# B&R Automation Studio project A2019059_Linka_Power_CP (part 39)

#### Main.st - Init, cyclic, exit code
```iecst
PROGRAM _INIT
	P34_Vizu.GoPage:= 'PageBootP34';

END_PROGRAM

PROGRAM _CYCLIC

	//************************************Filter alarmov**************************************************************//
	FilterVizu_P34:= '[{"logicalOperator":"and","value":300,"conditionType":">=","columnType":"cod","useAlarmState":false,"alarmState":0},{"value":500,"conditionType":"<=","columnType":"cod","useAlarmState":false,"alarmState":0}]';

	//***********************************Zobrazenie warningov pracoviska 3****************************************************//
	//0 - Pracovisko je vypnuté.
	//1 - Prebieha inicializácia pracoviska.
	//2 - Na pracovisku prebieha výroba.
	//3 - Prebieha ukončenie pracovného cyklu pracoviska.
	//4 - Prebieha režim vyprázdnenia linky.
	//5 - Doplň zásobník skrutiek K40 !!!
	//6 - Doplň zásobník skrutiek M5 !!!
	//7 - Niesu založené správne kontakty na HV teste !!!
	//8 - Niesu založené správne kontakty na Leakage teste stanica A !!!
	//9 - Niesu založené správne kontakty na Leakage teste stanica B !!!

	IF Linka.PAR.ZvolenyModel = '4F' AND NOT P3_Srobovanie.IN.HVTest_TypKonektoru_4F THEN
		P34_Vizu.WarningsP3_Index:= 7;
	ELSIF Linka.PAR.ZvolenyModel = '5F' AND NOT P3_Srobovanie.IN.HVTest_TypKonektoru_5F_5H THEN
		P34_Vizu.WarningsP3_Index:= 7;
	ELSIF Linka.PAR.ZvolenyModel = '5H' AND NOT P3_Srobovanie.IN.HVTest_TypKonektoru_5F_5H THEN
		P34_Vizu.WarningsP3_Index:= 7;
	ELSIF Linka.PAR.ZvolenyModel = '4F' AND NOT P3_LeakageTestA.IN.Tester_TypKonektoru_4F THEN
		P34_Vizu.WarningsP3_Index:= 8;
	ELSIF Linka.PAR.ZvolenyModel = '5F' AND NOT P3_LeakageTestA.IN.Tester_TypKonektoru_5F_5H THEN
		P34_Vizu.WarningsP3_Index:= 8;
	ELSIF Linka.PAR.ZvolenyModel = '5H' AND NOT P3_LeakageTestA.IN.Tester_TypKonektoru_5F_5H THEN
		P34_Vizu.WarningsP3_Index:= 8;
	ELSIF Linka.PAR.ZvolenyModel = '4F' AND NOT P3_LeakageTestB.IN.Tester_TypKonektoru_4F THEN
		P34_Vizu.WarningsP3_Index:= 9;
	ELSIF Linka.PAR.ZvolenyModel = '5F' AND NOT P3_LeakageTestB.IN.Tester_TypKonektoru_5F_5H THEN
		P34_Vizu.WarningsP3_Index:= 9;
	ELSIF Linka.PAR.ZvolenyModel = '5H' AND NOT P3_LeakageTestB.IN.Tester_TypKonektoru_5F_5H THEN
		P34_Vizu.WarningsP3_Index:= 9;
	ELSIF P3_Srobovanie.STAV.Zasobnik_K40_Prazdny THEN
		P34_Vizu.WarningsP3_Index:= 5;
	ELSIF P3_Srobovanie.STAV.Zasobnik_M5_Prazdny THEN
        P34_Vizu.WarningsP3_Index:= 6;
    ELSIF Linka.TestovaciKus THEN
        P34_Vizu.WarningsP3_Index:= 11;
	ELSIF Linka.VyprazdnenieLinky THEN
		P34_Vizu.WarningsP3_Index:= 4;
	ELSIF P3_Pracovisko.STAV.Automat AND NOT P3_Pracovisko.STAV.PoINIT AND NOT P3_Pracovisko.STAV.UkoncenieCyklu_BUSY THEN
		P34_Vizu.WarningsP3_Index:= 1;
	ELSIF P3_Pracovisko.STAV.PoINIT AND NOT P3_Pracovisko.STAV.UkoncenieCyklu_BUSY THEN
		P34_Vizu.WarningsP3_Index:= 2;
	ELSIF P3_Pracovisko.STAV.UkoncenieCyklu_BUSY THEN
		P34_Vizu.WarningsP3_Index:= 3;
	ELSIF NOT P3_Pracovisko.STAV.Automat THEN
		P34_Vizu.WarningsP3_Index:= 0;
	END_IF

	P34_Vizu.WarningsP3_Index;

	//************************Prepínanie farby textového pola warning pracoviska 3***********************************//
	IF P34_Vizu.WarningsP3_Index = 0 THEN
		P34_Vizu.WarningsP3_Farba:= "TextOutput_Green";
	ELSIF P34_Vizu.WarningsP3_Index = 1 THEN
		P34_Vizu.WarningsP3_Farba:= "TextOutput_Green";
	ELSIF P34_Vizu.WarningsP3_Index = 2 THEN
		P34_Vizu.WarningsP3_Farba:= "TextOutput_Green";
	ELSIF P34_Vizu.WarningsP3_Index = 3 THEN
		P34_Vizu.WarningsP3_Farba:= "TextOutput_Green";
	ELSIF P34_Vizu.WarningsP3_Index = 4 THEN
        P34_Vizu.WarningsP3_Farba:= "TextOutput_Green";
    ELSIF P34_Vizu.WarningsP3_Index = 11 THEN
        P34_Vizu.WarningsP3_Farba:= "TextOutput_Green";
	ELSE
		IF Blikac1s THEN
			P34_Vizu.WarningsP3_Farba:= "TextOutput_Red";
		ELSE
			P34_Vizu.WarningsP3_Farba:= "TextOutput_Grey";
		END_IF
	END_IF

	//***********************************Zobrazenie warningov pracoviska 4****************************************************//
	//0 - Pracovisko je vypnuté.
	//1 - Prebieha inicializácia pracoviska.
	//2 - Na pracovisku prebieha výroba.
	//3 - Prebieha ukončenie pracovného cyklu pracoviska.
	//4 - Prebieha režim vyprázdnenia linky.
	//5 - Niesu založené správne kontakty na Funkčnom teste stanica A !!!
	//6 - Niesu založené správne kontakty na Funkčnom teste stanica B !!!

	IF Linka.PAR.ZvolenyModel = '4F' AND NOT P4_FunkcnyTestA.IN.TypSpodnychKontaktov_4F THEN
		P34_Vizu.WarningsP4_Index:= 5;
	ELSIF Linka.PAR.ZvolenyModel = '5F' AND NOT P4_FunkcnyTestA.IN.TypSpodnychKontaktov_5F_5H THEN
		P34_Vizu.WarningsP4_Index:= 5;
	ELSIF Linka.PAR.ZvolenyModel = '5H' AND NOT P4_FunkcnyTestA.IN.TypSpodnychKontaktov_5F_5H THEN
		P34_Vizu.WarningsP4_Index:= 5;
	ELSIF Linka.PAR.ZvolenyModel = '4F' AND NOT P4_FunkcnyTestB.IN.TypSpodnychKontaktov_4F THEN
		P34_Vizu.WarningsP4_Index:= 6;
	ELSIF Linka.PAR.ZvolenyModel = '5F' AND NOT P4_FunkcnyTestB.IN.TypSpodnychKontaktov_5F_5H THEN
		P34_Vizu.WarningsP4_Index:= 6;
	ELSIF Linka.PAR.ZvolenyModel = '5H' AND NOT P4_FunkcnyTestB.IN.TypSpodnychKontaktov_5F_5H THEN
        P34_Vizu.WarningsP4_Index:= 6;
    ELSIF Linka.TestovaciKus THEN
        P34_Vizu.WarningsP4_Index:= 8;
	ELSIF Linka.VyprazdnenieLinky THEN
		P34_Vizu.WarningsP4_Index:= 4;
	ELSIF P4_Pracovisko.STAV.Automat AND NOT P4_Pracovisko.STAV.PoINIT AND NOT P4_Pracovisko.STAV.UkoncenieCyklu_BUSY THEN
		P34_Vizu.WarningsP4_Index:= 1;
	ELSIF P4_Pracovisko.STAV.PoINIT AND NOT P4_Pracovisko.STAV.UkoncenieCyklu_BUSY THEN
		P34_Vizu.WarningsP4_Index:= 2;
	ELSIF P4_Pracovisko.STAV.UkoncenieCyklu_BUSY THEN
		P34_Vizu.WarningsP4_Index:= 3;
	ELSIF NOT P4_Pracovisko.STAV.Automat THEN
		P34_Vizu.WarningsP4_Index:= 0;
	END_IF

	//************************Prepínanie farby textového pola warning pracoviska 4***********************************//
	IF P34_Vizu.WarningsP4_Index = 0 THEN
		P34_Vizu.WarningsP4_Farba:= "TextOutput_Green";
	ELSIF P34_Vizu.WarningsP4_Index = 1 THEN
		P34_Vizu.WarningsP4_Farba:= "TextOutput_Green";
	ELSIF P34_Vizu.WarningsP4_Index = 2 THEN
		P34_Vizu.WarningsP4_Farba:= "TextOutput_Green";
	ELSIF P34_Vizu.WarningsP4_Index = 3 THEN
		P34_Vizu.WarningsP4_Farba:= "TextOutput_Green";
	ELSIF P34_Vizu.WarningsP4_Index = 4 THEN
        P34_Vizu.WarningsP4_Farba:= "TextOutput_Green";
    ELSIF P34_Vizu.WarningsP4_Index = 8 THEN
        P34_Vizu.WarningsP4_Farba:= "TextOutput_Green";
	ELSE
		IF Blikac1s THEN
			P34_Vizu.WarningsP4_Farba:= "TextOutput_Red";
		ELSE
			P34_Vizu.WarningsP4_Farba:= "TextOutput_Grey";
		END_IF
	END_IF

	//***********************Prepnutie na obrazovku Automat z ručného režimu******************//
    IF P3_Pracovisko.STAV.Manual AND NOT Safety.STAV.P3_ZamkyBunky_AKTIVNE THEN
        P3_Pracovisko.Reset:= TRUE;
        P34_Vizu.GoPage:= 'PageBootP34';
    END_IF
    IF P4_Pracovisko.STAV.Manual AND NOT Safety.STAV.P4_ZamkyBunky_AKTIVNE THEN
        P4_Pracovisko.Reset:= TRUE;
        P34_Vizu.GoPage:= 'PageBootP34';
    END_IF

	//***********************Prepnutie bootovacej obrazovky********************************//
	IF NOT Safety.STAV.SafetyPLC_Nabehlo THEN
        P34_Vizu.GoPage:= 'PageBootP34';
    ELSIF CasPrepnutiaObrazovky.Q THEN
        P34_Vizu.GoPage:= 'PageBootP34';
	ELSIF P34_Vizu.ActualPage = 'PageBootP34' AND Safety.STAV.SafetyPLC_Nabehlo THEN
		P34_Vizu.GoPage:= 'PageAutomatP34';
	END_IF

    CasPrepnutiaObrazovky.IN:= P34_Vizu.ActualPage = 'PageBootP34' AND P34_Vizu.GoPage = 'PageAutomatP34';
    CasPrepnutiaObrazovky.PT:= T#5s;
    CasPrepnutiaObrazovky();

    //**************************Zamknutie editácie parametrov *********************************//

    IF P34_UrovenPrihlasenehoUzivatela >= 20 THEN
        P34_Vizu.EditaciaParametrov_ENABLE:= TRUE;
    ELSE
        P34_Vizu.EditaciaParametrov_ENABLE:= FALSE;
    END_IF

	//*************************************Zamknutie tlačítok - Pracovisko 3***************************************************************//
	//Tlačítko Štat Automat //
	IF P3_Pracovisko.STAV.UkoncenieCyklu_BUSY THEN
		P34_Vizu.TL_StartAutomat_ENABLE_P3:= FALSE;
	ELSIF P3_Pracovisko.STAV.PORUCHA THEN
		P34_Vizu.TL_StartAutomat_ENABLE_P3:= FALSE;
	ELSIF Linka.PAR.ZvolenyModel = '4F' AND NOT P3_Srobovanie.IN.HVTest_TypKonektoru_4F THEN
		P34_Vizu.TL_StartAutomat_ENABLE_P3:= FALSE;
	ELSIF Linka.PAR.ZvolenyModel = '5F' AND NOT P3_Srobovanie.IN.HVTest_TypKonektoru_5F_5H THEN
		P34_Vizu.TL_StartAutomat_ENABLE_P3:= FALSE;
	ELSIF Linka.PAR.ZvolenyModel = '5H' AND NOT P3_Srobovanie.IN.HVTest_TypKonektoru_5F_5H THEN
		P34_Vizu.TL_StartAutomat_ENABLE_P3:= FALSE;
	ELSIF Linka.PAR.ZvolenyModel = '4F' AND NOT P3_LeakageTestA.IN.Tester_TypKonektoru_4F THEN
		P34_Vizu.TL_StartAutomat_ENABLE_P3:= FALSE;
	ELSIF Linka.PAR.ZvolenyModel = '5F' AND NOT P3_LeakageTestA.IN.Tester_TypKonektoru_5F_5H THEN
		P34_Vizu.TL_StartAutomat_ENABLE_P3:= FALSE;
	ELSIF Linka.PAR.ZvolenyModel = '5H' AND NOT P3_LeakageTestA.IN.Tester_TypKonektoru_5F_5H THEN
		P34_Vizu.TL_StartAutomat_ENABLE_P3:= FALSE;
	ELSIF Linka.PAR.ZvolenyModel = '4F' AND NOT P3_LeakageTestB.IN.Tester_TypKonektoru_4F THEN
		P34_Vizu.TL_StartAutomat_ENABLE_P3:= FALSE;
	ELSIF Linka.PAR.ZvolenyModel = '5F' AND NOT P3_LeakageTestB.IN.Tester_TypKonektoru_5F_5H THEN
		P34_Vizu.TL_StartAutomat_ENABLE_P3:= FALSE;
	ELSIF Linka.PAR.ZvolenyModel = '5H' AND NOT P3_LeakageTestB.IN.Tester_TypKonektoru_5F_5H THEN
		P34_Vizu.TL_StartAutomat_ENABLE_P3:= FALSE;
	ELSIF NOT Safety.STAV.P3_ZonaBunky_AKTIVNA THEN
		P34_Vizu.TL_StartAutomat_ENABLE_P3:= FALSE;
	ELSE
		P34_Vizu.TL_StartAutomat_ENABLE_P3:= TRUE;
	END_IF

	//Tlačítko Ukončenie Cyklu//
	IF P3_Pracovisko.STAV.PoINIT THEN
		P34_Vizu.TL_KoniecCyklu_ENABLE_P3:= TRUE;
	ELSE
		P34_Vizu.TL_KoniecCyklu_ENABLE_P3:= FALSE;
	END_IF

    //Tlačítko STOP//
    IF P3_Pracovisko.STAV.PoINIT THEN
        P34_Vizu.TL_STOP_ENABLE_P3:= FALSE;
    ELSE
        P34_Vizu.TL_STOP_ENABLE_P3:= TRUE;
    END_IF

	//Tlačítko Režim Automat//

	P34_Vizu.TL_RezimAutomat_ENABLE:= TRUE;

	//Tlačítko Režim Manual - pracovisko 3//
	IF P3_Pracovisko.STAV.Automat THEN
		P34_Vizu.TL_RezimManual_ENABLE_P3:= FALSE;
	ELSIF NOT P3_Pracovisko.STAV.Manual AND NOT P3_Pracovisko.STAV.READY THEN
		P34_Vizu.TL_RezimManual_ENABLE_P3:= FALSE;
	ELSIF NOT Safety.STAV.P3_ZamkyBunky_AKTIVNE THEN
        P34_Vizu.TL_RezimManual_ENABLE_P3:= FALSE;
    ELSE
		P34_Vizu.TL_RezimManual_ENABLE_P3:= TRUE;
	END_IF

    //Tlačítka ovládania zámkov//
    IF NOT P3_Pracovisko.STAV.Automat THEN
        P34_Vizu.TL_OvladaniaZamkov_ENABLE_P3:= TRUE;
    ELSE
        P34_Vizu.TL_OvladaniaZamkov_ENABLE_P3:= FALSE;
    END_IF

    //Volba zapnutia Leakage Testu//
    IF P3_Pracovisko.STAV.Automat THEN
        P34_Vizu.VolbaLeakageTestu_ENABLE:= FALSE;
    ELSE
        P34_Vizu.VolbaLeakageTestu_ENABLE:= TRUE;
    END_IF

    //Tlačítka spustenie čistenie skrutkovačiek v ručnom režime//
    IF NOT P3_Srobovacky_VychodziaPozicia THEN
        P34_Vizu.RR_CistenieSkrutkovaciek_ENABLE:= FALSE;
    ELSIF P3_Srobovanie.STAV.Cistenie_K40_BUSY THEN
        P34_Vizu.RR_CistenieSkrutkovaciek_ENABLE:= FALSE;
    ELSIF NOT P3_Srobovanie.STAV.OsY_HomingOK THEN
        P34_Vizu.RR_CistenieSkrutkovaciek_ENABLE:= FALSE;
    ELSIF P34_UrovenPrihlasenehoUzivatela < 20 THEN
        P34_Vizu.RR_CistenieSkrutkovaciek_ENABLE:= FALSE;
    ELSIF P3_Srobovanie.RR_PolohujNaPoziciuSkrutky_4F5F THEN
        P34_Vizu.RR_CistenieSkrutkovaciek_ENABLE:= FALSE;
    ELSIF P3_Srobovanie.RR_PolohujNaPoziciuSkrutky_5H THEN
        P34_Vizu.RR_CistenieSkrutkovaciek_ENABLE:= FALSE;
    ELSE
        P34_Vizu.RR_CistenieSkrutkovaciek_ENABLE:= TRUE;
    END_IF

    //Tlačítka ovládania osy Y manipulatora šróbovačiek//
    IF NOT P3_Srobovanie.STAV.OsY_HomingOK THEN
        P34_Vizu.Srobovanie_OvlManipOsY_ENABLE:= FALSE;
    ELSIF NOT P3_Srobovacky_VychodziaPozicia THEN
        P34_Vizu.Srobovanie_OvlManipOsY_ENABLE:= FALSE;
    ELSIF P3_Srobovanie.RR_PolohujNaPoziciuSkrutky_4F5F THEN
        P34_Vizu.Srobovanie_OvlManipOsY_ENABLE:= FALSE;
    ELSIF P3_Srobovanie.RR_PolohujNaPoziciuSkrutky_5H THEN
        P34_Vizu.Srobovanie_OvlManipOsY_ENABLE:= FALSE;
    ELSIF P3_Srobovanie.STAV.Cistenie_K40_BUSY THEN
        P34_Vizu.Srobovanie_OvlManipOsY_ENABLE:= FALSE;
    ELSE
        P34_Vizu.Srobovanie_OvlManipOsY_ENABLE:= TRUE;
    END_IF

    //Zamknutie tlačítok test pozicii skrutkovačiek//
    IF NOT P3_Srobovanie.STAV.OsY_HomingOK THEN
        P34_Vizu.RR_PozicieSkrutiek_ENABLE:= FALSE;
    ELSIF NOT P3_Srobovacky_VychodziaPozicia THEN
        P34_Vizu.RR_PozicieSkrutiek_ENABLE:= FALSE;
    ELSIF P3_Srobovanie.STAV.Cistenie_K40_BUSY THEN
        P34_Vizu.RR_PozicieSkrutiek_ENABLE:= FALSE;
    ELSIF P34_UrovenPrihlasenehoUzivatela < 100 THEN
        P34_Vizu.RR_PozicieSkrutiek_ENABLE:= FALSE;
    ELSIF P3_Srobovanie.RR_PolohujNaPoziciuSkrutky_4F5F THEN
        P34_Vizu.RR_PozicieSkrutiek_ENABLE:= FALSE;
    ELSIF P3_Srobovanie.RR_PolohujNaPoziciuSkrutky_5H THEN
        P34_Vizu.RR_PozicieSkrutiek_ENABLE:= FALSE;
    ELSE
        P34_Vizu.RR_PozicieSkrutiek_ENABLE:= TRUE;
    END_IF

    //Tlačítko testovania Leakage Testu A v ručnom režime//
    IF NOT Safety.STAV.P3_ZonaBunky_AKTIVNA THEN
        P34_Vizu.LeakageTestA_Testovanie_ENABLE:= FALSE;
    ELSIF NOT P3_LeakageTestA.IN.PritomnostPaletky_S23 THEN
       P34_Vizu.LeakageTestA_Testovanie_ENABLE:= FALSE;
    ELSE
        P34_Vizu.LeakageTestA_Testovanie_ENABLE:= TRUE;
    END_IF

    //Tlačítko testovania Leakage Testu B v ručnom režime//
    IF NOT Safety.STAV.P3_ZonaBunky_AKTIVNA THEN
        P34_Vizu.LeakageTestB_Testovanie_ENABLE:= FALSE;
    ELSIF NOT P3_LeakageTestB.IN.PritomnostPaletky_S24 THEN
        P34_Vizu.LeakageTestB_Testovanie_ENABLE:= FALSE;
    ELSE
        P34_Vizu.LeakageTestB_Testovanie_ENABLE:= TRUE;
    END_IF

    //Zamknutie tlačítok ovládania Leakage testu A v ručnom režime//
    IF P3_LeakageTestA.STAV.TestovaciaSekvencia_BUSY THEN
        P34_Vizu.LeakageTestA_RR_ENABLE:= FALSE;
    ELSE
        P34_Vizu.LeakageTestA_RR_ENABLE:= TRUE;
    END_IF

   //Zamknutie tlačítok ovládania Leakage testu B v ručnom režime//
    IF P3_LeakageTestB.STAV.TestovaciaSekvencia_BUSY THEN
        P34_Vizu.LeakageTestB_RR_ENABLE:= FALSE;
    ELSE
        P34_Vizu.LeakageTestB_RR_ENABLE:= TRUE;
    END_IF

	//*************************************Zamknutie tlačítok - Pracovisko 4***************************************************************//
	//Tlačítko Štat Automat//
	IF P4_Pracovisko.STAV.UkoncenieCyklu_BUSY THEN
		P34_Vizu.TL_StartAutomat_ENABLE_P4:= FALSE;
	ELSIF P4_Pracovisko.STAV.PORUCHA THEN
		P34_Vizu.TL_StartAutomat_ENABLE_P4:= FALSE;
	ELSIF Linka.PAR.ZvolenyModel = '4F' AND NOT P4_FunkcnyTestA.IN.TypSpodnychKontaktov_4F THEN
		P34_Vizu.TL_StartAutomat_ENABLE_P4:= FALSE;
	ELSIF Linka.PAR.ZvolenyModel = '5F' AND NOT P4_FunkcnyTestA.IN.TypSpodnychKontaktov_5F_5H THEN
		P34_Vizu.TL_StartAutomat_ENABLE_P4:= FALSE;
	ELSIF Linka.PAR.ZvolenyModel = '5H' AND NOT P4_FunkcnyTestA.IN.TypSpodnychKontaktov_5F_5H THEN
		P34_Vizu.TL_StartAutomat_ENABLE_P4:= FALSE;
	ELSIF Linka.PAR.ZvolenyModel = '4F' AND NOT P4_FunkcnyTestB.IN.TypSpodnychKontaktov_4F THEN
		P34_Vizu.TL_StartAutomat_ENABLE_P4:= FALSE;
	ELSIF Linka.PAR.ZvolenyModel = '5F' AND NOT P4_FunkcnyTestB.IN.TypSpodnychKontaktov_5F_5H THEN
		P34_Vizu.TL_StartAutomat_ENABLE_P4:= FALSE;
	ELSIF Linka.PAR.ZvolenyModel = '5H' AND NOT P4_FunkcnyTestB.IN.TypSpodnychKontaktov_5F_5H THEN
		P34_Vizu.TL_StartAutomat_ENABLE_P4:= FALSE;
	ELSIF NOT Safety.STAV.P4_ZonaBunky_AKTIVNA THEN
		P34_Vizu.TL_StartAutomat_ENABLE_P4:= FALSE;
	ELSE
		P34_Vizu.TL_StartAutomat_ENABLE_P4:= TRUE;
	END_IF

	//Tlačítko Ukončenie Cyklu//
	IF P4_Pracovisko.STAV.PoINIT THEN
		P34_Vizu.TL_KoniecCyklu_ENABLE_P4:= TRUE;
	ELSE
		P34_Vizu.TL_KoniecCyklu_ENABLE_P4:= FALSE;
	END_IF

    //Tlačítko STOP//
    IF P4_Pracovisko.STAV.PoINIT THEN
        P34_Vizu.TL_STOP_ENABLE_P4:= FALSE;
    ELSE
        P34_Vizu.TL_STOP_ENABLE_P4:= TRUE;
    END_IF

    //Tlačítko vyprázdnenie linky//
    IF Linka.VyprazdnenieLinky THEN
        P34_Vizu.TL_VyprazdnenieLinky_ENABLE:= FALSE;
    ELSIF NOT P4_Pracovisko.STAV.Automat THEN
        P34_Vizu.TL_VyprazdnenieLinky_ENABLE:= FALSE;
    ELSIF Linka.TestovaciKus THEN
        P34_Vizu.TL_VyprazdnenieLinky_ENABLE:= FALSE;
    ELSE
        P34_Vizu.TL_VyprazdnenieLinky_ENABLE:= TRUE;
    END_IF

	//Tlačítka ovládania zámkov//
	IF NOT P4_Pracovisko.STAV.Automat THEN
		P34_Vizu.TL_OvladaniaZamkov_ENABLE_P4:= TRUE;
	ELSE
		P34_Vizu.TL_OvladaniaZamkov_ENABLE_P4:= FALSE;
	END_IF

    //Tlačítko Režim Manual - pracovisko 4//
    IF P4_Pracovisko.STAV.Automat THEN
        P34_Vizu.TL_RezimManual_ENABLE_P4:= FALSE;
    ELSIF NOT P4_Pracovisko.STAV.Manual AND NOT P4_Pracovisko.STAV.READY THEN
        P34_Vizu.TL_RezimManual_ENABLE_P4:= FALSE;
    ELSIF NOT Safety.STAV.P4_ZamkyBunky_AKTIVNE THEN
        P34_Vizu.TL_RezimManual_ENABLE_P4:= FALSE;
    ELSE
        P34_Vizu.TL_RezimManual_ENABLE_P4:= TRUE;
    END_IF

    //Volba zapnutia Funkčného Testu//
    IF P4_Pracovisko.STAV.Automat THEN
        P34_Vizu.VolbaFunkcnehoTestu_ENABLE:= FALSE;
    ELSE
        P34_Vizu.VolbaFunkcnehoTestu_ENABLE:= TRUE;
    END_IF

    //Tlačítko testovania Funkčného Testu A v ručnom režime//
    IF NOT Safety.STAV.P4_ZonaBunky_AKTIVNA THEN
        P34_Vizu.FunkcnyTestA_Testovanie_ENABLE:= FALSE;
    ELSIF NOT P4_FunkcnyTestA.IN.PritomnostPaletky_S10 THEN
        P34_Vizu.FunkcnyTestA_Testovanie_ENABLE:= FALSE;
    ELSE
        P34_Vizu.FunkcnyTestA_Testovanie_ENABLE:= TRUE;
    END_IF

    //Tlačítko testovania Funkčného Testu B v ručnom režime//
    IF NOT Safety.STAV.P4_ZonaBunky_AKTIVNA THEN
        P34_Vizu.FunkcnyTestB_Testovanie_ENABLE:= FALSE;
    ELSIF NOT P4_FunkcnyTestB.IN.PritomnostPaletky_S11 THEN
        P34_Vizu.FunkcnyTestB_Testovanie_ENABLE:= FALSE;
    ELSE
        P34_Vizu.FunkcnyTestB_Testovanie_ENABLE:= TRUE;
    END_IF

    //Tlačítka ovládania výťahu v ručnom režime//
    IF NOT P4_Vytah.STAV.ServoZdvihu_HomingOK THEN
        P34_Vizu.TL_OvladanieVytahu_ENABLE:= FALSE;
    ELSIF P4_Vytah.STAV.ServoZdvihu_Homing_BUSY THEN
        P34_Vizu.TL_OvladanieVytahu_ENABLE:= FALSE;
    ELSIF P4_Vytah.IN.VystupDopravnikaVytahu_OS11 THEN
        P34_Vizu.TL_OvladanieVytahu_ENABLE:= FALSE;
    ELSIF NOT Safety.STAV.P4_Vytah_Bariera_AKTIVNA THEN
        P34_Vizu.TL_OvladanieVytahu_ENABLE:= FALSE;
    ELSE
        P34_Vizu.TL_OvladanieVytahu_ENABLE:= TRUE;
    END_IF

    //Tlačítko homing zdvihu výťahu//
    IF P4_Vytah.IN.VystupDopravnikaVytahu_OS11 THEN
        P34_Vizu.TL_HomingVytahu_ENABLE:= FALSE;
    ELSIF NOT Safety.STAV.P4_Vytah_Bariera_AKTIVNA THEN
        P34_Vizu.TL_HomingVytahu_ENABLE:= FALSE;
    ELSE
        P34_Vizu.TL_HomingVytahu_ENABLE:= TRUE;
    END_IF

    //Tlačítka ovládania zdvihu aplikátora etikety v ručnom režime//
    IF NOT P4_Etiketovacka.STAV.ServoZdvihu_HomingOK THEN
        P34_Vizu.TL_OvlZdvihuAplikEtikety_ENABLE:= FALSE;
    ELSIF NOT P4_Etiketovacka.IN.Aplikator_ZASUNUTY_MS35 THEN
        P34_Vizu.TL_OvlZdvihuAplikEtikety_ENABLE:= FALSE;
    ELSIF P4_Etiketovacka.IN.PritlakPaskyOdisteny_IS84 THEN
        P34_Vizu.TL_OvlZdvihuAplikEtikety_ENABLE:= FALSE;
    ELSE
        P34_Vizu.TL_OvlZdvihuAplikEtikety_ENABLE:= TRUE;
    END_IF

    //Tlačítko testovania Etiketovania v ručnom režime//
    IF NOT Safety.STAV.P4_ZonaBunky_AKTIVNA THEN
        P34_Vizu.Etiketovacka_Testovanie_ENABLE:= FALSE;
    ELSIF NOT P4_Etiketovacka.IN.PritomnostPaletky_S12 THEN
        P34_Vizu.Etiketovacka_Testovanie_ENABLE:= FALSE;
    ELSIF NOT P4_Etiketovacka.STAV.ServoZdvihu_HomingOK THEN
        P34_Vizu.Etiketovacka_Testovanie_ENABLE:= FALSE;
    ELSIF P4_Etiketovacka.IN.PritlakPaskyOdisteny_IS84 THEN
        P34_Vizu.Etiketovacka_Testovanie_ENABLE:= FALSE;
    ELSE
        P34_Vizu.Etiketovacka_Testovanie_ENABLE:= TRUE;
    END_IF

    //***************************************Zmena farieb tlačítok pre ovládanie zámkou - Pracovisko 3********************************//
    //Predné dvere pravá strana//
	IF Safety.OUT.P3_ZamkniZamok_PredneDverePS AND Safety.IN.P3_PredneDverePS_PritomPetlice THEN
		P34_Vizu.TL_PrednyZamokPS_Farba_P3:= "Button_Green";
	ELSIF Safety.IN.P3_PredneDverePS_PritomPetlice THEN
		IF Blikac1s THEN
			P34_Vizu.TL_PrednyZamokPS_Farba_P3:= "Button_Blue";
		ELSE
			P34_Vizu.TL_PrednyZamokPS_Farba_P3:= "Operate";
		END_IF
	ELSE
		P34_Vizu.TL_PrednyZamokPS_Farba_P3:= "Button_Red";
	END_IF

	//Predné dvere lavá strana//
	IF Safety.OUT.P3_ZamkniZamok_PredneDvereLS AND Safety.IN.P3_PredneDvereLS_PritomPetlice THEN
		P34_Vizu.TL_PrednyZamokLS_Farba_P3:= "Button_Green";
	ELSIF Safety.IN.P3_PredneDvereLS_PritomPetlice THEN
		IF Blikac1s THEN
			P34_Vizu.TL_PrednyZamokLS_Farba_P3:= "Button_Blue";
		ELSE
			P34_Vizu.TL_PrednyZamokLS_Farba_P3:= "Operate";
		END_IF
	ELSE
		P34_Vizu.TL_PrednyZamokLS_Farba_P3:= "Button_Red";
	END_IF

	//Zadné dvere //
	IF Safety.OUT.P3_ZamkniZamok_ZadneDvere AND Safety.IN.P3_ZadneDvere_PritomPetlice THEN
		P34_Vizu.TL_ZadnyZamok_Farba_P3:= "Button_Green";
	ELSIF Safety.IN.P3_ZadneDvere_PritomPetlice THEN
		IF Blikac1s THEN
			P34_Vizu.TL_ZadnyZamok_Farba_P3:= "Button_Blue";
		ELSE
			P34_Vizu.TL_ZadnyZamok_Farba_P3:= "Operate";
		END_IF
	ELSE
		P34_Vizu.TL_ZadnyZamok_Farba_P3:= "Button_Red";
	END_IF

	//***************************************Zmena farieb tlačítok pre ovládanie zámkou - Pracovisko 4********************************//
	//Predné dvere //
	IF Safety.OUT.P4_ZamkniZamok_PredneDvere AND Safety.IN.P4_PredneDvere_PritomPetlice THEN
		P34_Vizu.TL_PrednyZamok_Farba_P4:= "Button_Green";
	ELSIF Safety.IN.P4_PredneDvere_PritomPetlice THEN
		IF Blikac1s THEN
			P34_Vizu.TL_PrednyZamok_Farba_P4:= "Button_Blue";
		ELSE
			P34_Vizu.TL_PrednyZamok_Farba_P4:= "Operate";
		END_IF
	ELSE
		P34_Vizu.TL_PrednyZamok_Farba_P4:= "Button_Red";
	END_IF

	//***********************************Prepínanie stavov pracovísk - Pracovisko 3*******************************************************************//
	//Dopravníky//
	IF NOT P3_Dopravniky.IN.HornyDoprav_READY OR NOT P3_Dopravniky.IN.SpodnyDoprav_READY THEN
		P34_Vizu.IndexStavu_DopravnikP3:= 3;
	ELSIF P3_Dopravniky.Automat AND NOT P3_Dopravniky.STAV.PoINIT THEN
		P34_Vizu.IndexStavu_DopravnikP3:= 1;
	ELSIF P3_Dopravniky.Automat AND P3_Dopravniky.STAV.PoINIT THEN
		P34_Vizu.IndexStavu_DopravnikP3:= 2;
	ELSE
		P34_Vizu.IndexStavu_DopravnikP3:= 0;
	END_IF

	//Spodný stoper//
	IF P3_SpodnyStoper.Automat AND NOT P3_SpodnyStoper.STAV.PoINIT THEN
		P34_Vizu.IndexStavu_SpodnyStoperP3:= 1;
	ELSIF P3_SpodnyStoper.Automat AND P3_SpodnyStoper.STAV.PoINIT THEN
		P34_Vizu.IndexStavu_SpodnyStoperP3:= 2;
	ELSE
		P34_Vizu.IndexStavu_SpodnyStoperP3:= 0;
	END_IF

    //Vstupný stoper//
    IF P3_VstupnyStoper.Automat AND NOT P3_VstupnyStoper.STAV.PoINIT THEN
        P34_Vizu.IndexStavu_VstupnyStoper:= 1;
    ELSIF P3_VstupnyStoper.Automat AND P3_VstupnyStoper.STAV.PoINIT THEN
        P34_Vizu.IndexStavu_VstupnyStoper:= 2;
    ELSE
        P34_Vizu.IndexStavu_VstupnyStoper:= 0;
    END_IF

	//Stoper šrobovania//
	IF P3_PoruchaST1 THEN
		P34_Vizu.IndexStavu_StoperSrobovaniaP3:= 3;
	ELSIF P3_StoperSrobovania.Automat AND NOT P3_StoperSrobovania.STAV.PoINIT THEN
		P34_Vizu.IndexStavu_StoperSrobovaniaP3:= 1;
	ELSIF P3_StoperSrobovania.Automat AND P3_StoperSrobovania.STAV.PoINIT THEN
		P34_Vizu.IndexStavu_StoperSrobovaniaP3:= 2;
	ELSE
		P34_Vizu.IndexStavu_StoperSrobovaniaP3:= 0;
	END_IF

	//Šrobovanie//
	IF P3_PoruchaST1 THEN
		P34_Vizu.IndexStavu_SrobovanieP3:= 3;
	ELSIF P3_Srobovanie.Automat AND NOT P3_Srobovanie.STAV.PoINIT THEN
		P34_Vizu.IndexStavu_SrobovanieP3:= 1;
	ELSIF P3_Srobovanie.Automat AND P3_Srobovanie.STAV.PoINIT THEN
		P34_Vizu.IndexStavu_SrobovanieP3:= 2;
	ELSE
		P34_Vizu.IndexStavu_SrobovanieP3:= 0;
	END_IF

	//Akumulačný stoper//
	IF P3_AkumulacnyStoper.Automat AND NOT P3_AkumulacnyStoper.STAV.PoINIT THEN
		P34_Vizu.IndexStavu_AkumulacnyStoperP3:= 1;
	ELSIF P3_AkumulacnyStoper.Automat AND P3_AkumulacnyStoper.STAV.PoINIT THEN
		P34_Vizu.IndexStavu_AkumulacnyStoperP3:= 2;
	ELSE
		P34_Vizu.IndexStavu_AkumulacnyStoperP3:= 0;
	END_IF

	//Stoper Leakage Test A//
	IF P3_PoruchaST2 THEN
		P34_Vizu.IndexStavu_StoperLeakageTestA:= 3;
	ELSIF P3_LeakageTestA.Automat AND NOT P3_LeakageTestA.STAV.PoINIT THEN
		P34_Vizu.IndexStavu_StoperLeakageTestA:= 1;
	ELSIF P3_LeakageTestA.Automat AND P3_LeakageTestA.STAV.PoINIT THEN
		P34_Vizu.IndexStavu_StoperLeakageTestA:= 2;
	ELSE
		P34_Vizu.IndexStavu_StoperLeakageTestA:= 0;
	END_IF

	//Stoper Leakage Test B//
	IF P3_PoruchaST3 THEN
		P34_Vizu.IndexStavu_StoperLeakageTestB:= 3;
	ELSIF P3_LeakageTestB.Automat AND NOT P3_LeakageTestB.STAV.PoINIT THEN
		P34_Vizu.IndexStavu_StoperLeakageTestB:= 1;
	ELSIF P3_LeakageTestB.Automat AND P3_LeakageTestB.STAV.PoINIT THEN
		P34_Vizu.IndexStavu_StoperLeakageTestB:= 2;
	ELSE
		P34_Vizu.IndexStavu_StoperLeakageTestB:= 0;
	END_IF

	//***********************************Prepínanie stavov pracovísk - Pracovisko 4*******************************************************************//
	//Dopravníky//
	IF NOT P4_Dopravniky.IN.HornyDoprav_READY OR NOT P4_Dopravniky.IN.SpodnyDoprav_READY THEN
		P34_Vizu.IndexStavu_DopravnikP4:= 3;
	ELSIF P4_Dopravniky.Automat AND NOT P4_Dopravniky.STAV.PoINIT THEN
		P34_Vizu.IndexStavu_DopravnikP4:= 1;
	ELSIF P4_Dopravniky.Automat AND P4_Dopravniky.STAV.PoINIT THEN
		P34_Vizu.IndexStavu_DopravnikP4:= 2;
	ELSE
		P34_Vizu.IndexStavu_DopravnikP4:= 0;
	END_IF

	//Výťah//
	IF NOT P4_Vytah.IN.Dopravnik_READY THEN
		P34_Vizu.IndexStavu_Vytah:= 3;
	ELSIF P4_PoruchaST4 THEN
		P34_Vizu.IndexStavu_Vytah:= 3;
	ELSIF P4_Vytah.Automat AND NOT P4_Vytah.STAV.PoINIT THEN
		P34_Vizu.IndexStavu_Vytah:= 1;
	ELSIF P4_Vytah.Automat AND P4_Vytah.STAV.PoINIT THEN
		P34_Vizu.IndexStavu_Vytah:= 2;
	ELSE
		P34_Vizu.IndexStavu_Vytah:= 0;
	END_IF

	//Stoper Funkčný Test A//
	IF P4_PoruchaST1 THEN
		P34_Vizu.IndexStavu_StoperFunkcnyTestA:= 3;
	ELSIF P4_FunkcnyTestA.Automat AND NOT P4_FunkcnyTestA.STAV.PoINIT THEN
		P34_Vizu.IndexStavu_StoperFunkcnyTestA:= 1;
	ELSIF P4_FunkcnyTestA.Automat AND P4_FunkcnyTestA.STAV.PoINIT THEN
		P34_Vizu.IndexStavu_StoperFunkcnyTestA:= 2;
	ELSE
		P34_Vizu.IndexStavu_StoperFunkcnyTestA:= 0;
	END_IF

	//Stoper Funkčný Test B//
	IF P4_PoruchaST2 THEN
		P34_Vizu.IndexStavu_StoperFunkcnyTestB:= 3;
	ELSIF P4_FunkcnyTestB.Automat AND NOT P4_FunkcnyTestB.STAV.PoINIT THEN
		P34_Vizu.IndexStavu_StoperFunkcnyTestB:= 1;
	ELSIF P4_FunkcnyTestB.Automat AND P4_FunkcnyTestB.STAV.PoINIT THEN
		P34_Vizu.IndexStavu_StoperFunkcnyTestB:= 2;
	ELSE
		P34_Vizu.IndexStavu_StoperFunkcnyTestB:= 0;
	END_IF

	//Stoper Etiketovačky//
	IF P4_PoruchaST3 THEN
		P34_Vizu.IndexStavu_StoperEtiketovackyP4:= 3;
	ELSIF P4_Etiketovacka.Automat AND NOT P4_Etiketovacka.STAV.PoINIT THEN
		P34_Vizu.IndexStavu_StoperEtiketovackyP4:= 1;
	ELSIF P4_Etiketovacka.Automat AND P4_Etiketovacka.STAV.PoINIT THEN
		P34_Vizu.IndexStavu_StoperEtiketovackyP4:= 2;
	ELSE
		P34_Vizu.IndexStavu_StoperEtiketovackyP4:= 0;
	END_IF

END_PROGRAM

PROGRAM _EXIT
	(* Insert code here *)

END_PROGRAM
```

#### Variables.var - Local variables
```iecst
VAR
	CasPrepnutiaObrazovky : TON;
END_VAR
```

### Program Logical/Program/Pracovisko_3/P3_OvladanieSafety (IEC)

#### Main.st - Init, cyclic, exit code
```iecst
PROGRAM _INIT
	(* Insert code here *)

END_PROGRAM

PROGRAM _CYCLIC

    //******************************************Ovládanie zámkov dverí bunky****************************************//
    //Predné dvere - pravá strana//
	IF EDGEPOS(P34_Vizu.TL_ZamkniPrednyZamokPS_P3) THEN
		IF NOT Safety.OUT.P3_ZamkniZamok_PredneDverePS AND Safety.IN.P3_PredneDverePS_PritomPetlice THEN
            Safety.OUT.P3_ZamkniZamok_PredneDverePS:= TRUE;
        ELSIF Safety.OUT.P3_ZamkniZamok_PredneDverePS THEN
            Safety.OUT.P3_ZamkniZamok_PredneDverePS:= FALSE;
        END_IF
        P34_Vizu.TL_ZamkniPrednyZamokPS_P3:= FALSE;
    END_IF

    //Predné dvere - lavá strana//
    IF EDGEPOS(P34_Vizu.TL_ZamkniPrednyZamokLS_P3) THEN
        IF NOT Safety.OUT.P3_ZamkniZamok_PredneDvereLS AND Safety.IN.P3_PredneDvereLS_PritomPetlice THEN
            Safety.OUT.P3_ZamkniZamok_PredneDvereLS:= TRUE;
        ELSIF Safety.OUT.P3_ZamkniZamok_PredneDvereLS THEN
            Safety.OUT.P3_ZamkniZamok_PredneDvereLS:= FALSE;
        END_IF
        P34_Vizu.TL_ZamkniPrednyZamokLS_P3:= FALSE;
    END_IF

    //Zadné dvere//
    IF EDGEPOS(P34_Vizu.TL_ZamkniZadnyZamok_P3) THEN
        IF NOT Safety.OUT.P3_ZamkniZamok_ZadneDvere AND Safety.IN.P3_ZadneDvere_PritomPetlice THEN
            Safety.OUT.P3_ZamkniZamok_ZadneDvere:= TRUE;
        ELSIF Safety.OUT.P3_ZamkniZamok_ZadneDvere THEN
            Safety.OUT.P3_ZamkniZamok_ZadneDvere:= FALSE;
        END_IF
        P34_Vizu.TL_ZamkniZadnyZamok_P3:= FALSE;
    END_IF

	//Rset zóny bunky//
	CasResetZonyBunky.IN:= NOT Safety.STAV.P3_ZonaBunky_AKTIVNA	AND Safety.STAV.ZonaCS_AKTIVNA AND Safety.STAV.P3_ZamkyBunky_AKTIVNE AND (Safety.STAV.P3_VstupBunky_Bariera_AKTIVNA OR Safety.STAV.P2_ZamkyBunky_AKTIVNE) AND (Safety.STAV.P3_VystupBunky_Bariera_AKTIVNA OR Safety.STAV.P4_ZamkyBunky_AKTIVNE);

	IF CasResetZonyBunky.Q THEN
		Safety.IN.P3_ZonaBunky_RESET:= TRUE;
	ELSE
		Safety.IN.P3_ZonaBunky_RESET:= FALSE;
	END_IF

	CasResetZonyBunky.PT:= T#1s;
	CasResetZonyBunky();

END_PROGRAM

PROGRAM _EXIT
	(* Insert code here *)

END_PROGRAM
```

#### Variables.var - Local variables
```iecst
VAR
	CasResetZonyBunky : TON;
END_VAR
```

### Program Logical/Program/Pracovisko_4/P4_Main (IEC)

#### Main.st - Init, cyclic, exit code
```iecst
PROGRAM _INIT
	(* Insert code here *)

END_PROGRAM

PROGRAM _CYCLIC

	//Volanie podprogramu//
    OvlVentilovychTerminalov;
    ProfinetKomunikaciaKAM14;
    ProfinetKomunikaciaKAM15;
    ProfinetKomunikaciaKAM16;

    //******************************Stav moduly OK**************************************//
    IF P4_Pracovisko.STAV.ModulDI41_OK AND
        P4_Pracovisko.STAV.ModulDI42_OK AND
        P4_Pracovisko.STAV.ModulDM41_OK AND
        P4_Pracovisko.STAV.ModulDS41_OK AND
        P4_Pracovisko.STAV.ModulDS42_OK AND
        P4_Pracovisko.STAV.ModulSI41_OK AND
        P4_Pracovisko.STAV.ModulSI42_OK THEN
        P4_Pracovisko.STAV.Moduly_OK:= TRUE;
    ELSE
        P4_Pracovisko.STAV.Moduly_OK:= FALSE;
    END_IF

    //******************************Stav kamery OK**************************************//
    IF Linka.STAV.WenglorControlUnit_OK AND
        CAM14.STAV.READY THEN
        P4_Pracovisko.STAV.Kamery_OK:= TRUE;
    ELSE
        P4_Pracovisko.STAV.Kamery_OK:= FALSE;
    END_IF

    //******************************Stav ventilové terminály OK***************************//
    IF P4_Pracovisko.STAV.VentilovyTerminal_VT8_OK THEN
        P4_Pracovisko.STAV.VentiloveTerminaly_OK:= TRUE;
    ELSE
        P4_Pracovisko.STAV.VentiloveTerminaly_OK:= FALSE;
    END_IF

    //Ukončenie cyklu//
    IF P4_Pracovisko.KoniecCyklu THEN
        IF P4_Dopravniky.Automat THEN
            P4_Dopravniky.KoniecCyklu:= TRUE;
        END_IF
        IF P4_Vytah.Automat THEN
            P4_Vytah.KoniecCyklu:= TRUE;
        END_IF
        IF P4_FunkcnyTestA.Automat THEN
            P4_FunkcnyTestA.KoniecCyklu:= TRUE;
        END_IF
        IF P4_FunkcnyTestB.Automat THEN
            P4_FunkcnyTestB.KoniecCyklu:= TRUE;
        END_IF
        IF P4_Etiketovacka.Automat THEN
            P4_Etiketovacka.KoniecCyklu:= TRUE;
        END_IF
        P4_Pracovisko.KoniecCyklu:= FALSE;
    END_IF

    //Ukončenie cyklu pri poruche//
    IF EDGEPOS(P4_PoruchaST1) THEN
        IF P4_FunkcnyTestB.Automat THEN
            P4_FunkcnyTestB.KoniecCyklu:= TRUE;
        END_IF
        IF P4_Etiketovacka.Automat THEN
            P4_Etiketovacka.KoniecCyklu:= TRUE;
        END_IF
        IF P4_Dopravniky.Automat THEN
            P4_Dopravniky.KoniecCyklu:= TRUE;
        END_IF
    ELSIF EDGEPOS(P4_PoruchaST2) THEN
        IF P4_FunkcnyTestA.Automat THEN
            P4_FunkcnyTestA.KoniecCyklu:= TRUE;
        END_IF
        IF P4_Etiketovacka.Automat THEN
            P4_Etiketovacka.KoniecCyklu:= TRUE;
        END_IF
        IF P4_Dopravniky.Automat THEN
            P4_Dopravniky.KoniecCyklu:= TRUE;
        END_IF
    ELSIF EDGEPOS(P4_PoruchaST3) THEN
        IF P4_FunkcnyTestA.Automat THEN
            P4_FunkcnyTestA.KoniecCyklu:= TRUE;
        END_IF
        IF P4_FunkcnyTestB.Automat THEN
            P4_FunkcnyTestB.KoniecCyklu:= TRUE;
        END_IF
        IF P4_Dopravniky.Automat THEN
            P4_Dopravniky.KoniecCyklu:= TRUE;
        END_IF
    END_IF

    //Status prebieha ukončenie cyklu//
    IF P4_Dopravniky.KoniecCyklu OR
        P4_Vytah.KoniecCyklu OR
        P4_FunkcnyTestA.KoniecCyklu OR
        P4_FunkcnyTestB.KoniecCyklu OR
        P4_Etiketovacka.KoniecCyklu THEN
        P4_Pracovisko.STAV.UkoncenieCyklu_BUSY:= TRUE;
    ELSE
        P4_Pracovisko.STAV.UkoncenieCyklu_BUSY:= FALSE;
    END_IF

    //Resetovanie pracoviska//
    IF P4_Pracovisko.Reset THEN
        P4_Dopravniky.Reset:= TRUE;
        P4_Vytah.Reset:= TRUE;
        P4_FunkcnyTestA.Reset:= TRUE;
        P4_FunkcnyTestB.Reset:= TRUE;
        P4_Etiketovacka.Reset:= TRUE;
        P4_Pracovisko.Reset:= FALSE;
    END_IF

    //Prepnutie pracoviska do manualneho režimu//
    IF P4_Pracovisko.Manual THEN
        P4_Dopravniky.Manual:= TRUE;
        P4_Vytah.Manual:= TRUE;
        P4_FunkcnyTestA.Manual:= TRUE;
        P4_FunkcnyTestB.Manual:= TRUE;
        P4_Etiketovacka.Manual:= TRUE;
        P4_Pracovisko.Manual:= FALSE;
    END_IF

    //Spustenie pracoviska v automatickom režime//
    IF P4_Pracovisko.Automat THEN
        P4_Dopravniky.Automat:= TRUE;
        P4_Vytah.Automat:= TRUE;
        P4_FunkcnyTestA.Automat:= TRUE;
        P4_FunkcnyTestB.Automat:= TRUE;
        P4_Etiketovacka.Automat:= TRUE;
        P4_Pracovisko.Automat:= FALSE;
    END_IF

    //*********************************Príznaky pracoviska*******************************************//
    //Príznak pracovisko stav AUTOMAT//
    IF P4_Dopravniky.Automat OR
        P4_Vytah.Automat OR
        P4_FunkcnyTestA.Automat OR
        P4_FunkcnyTestB.Automat OR
        P4_Etiketovacka.Automat THEN
        P4_Pracovisko.STAV.Automat:= TRUE;
    ELSE
        P4_Pracovisko.STAV.Automat:= FALSE;
    END_IF

    //Priznak pracovisko stav MANUAL//
    IF P4_Dopravniky.Manual OR
        P4_Vytah.Manual OR
        P4_FunkcnyTestA.Manual OR
        P4_FunkcnyTestB.Manual OR
        P4_Etiketovacka.Manual THEN
        P4_Pracovisko.STAV.Manual:= TRUE;
    ELSE
        P4_Pracovisko.STAV.Manual:= FALSE;
    END_IF

    //Príznak pracovisko stav PoINIT//
    IF P4_Dopravniky.STAV.PoINIT AND
        (P4_Vytah.STAV.PoINIT OR NOT P4_Vytah.Automat) AND
        P4_FunkcnyTestA.STAV.PoINIT AND
        P4_FunkcnyTestB.STAV.PoINIT AND
        P4_Etiketovacka.STAV.PoINIT THEN
        P4_Pracovisko.STAV.PoINIT:= TRUE;
    ELSE
        P4_Pracovisko.STAV.PoINIT:= FALSE;
    END_IF

    //Príznak pracovisko stav READY//
    IF SC_P4_Dopravniky.Step = 1 AND
        SC_P4_Vytah.Step = 1 AND
        SC_P4_FunkcnyTestA.Step = 1 AND
        SC_P4_FunkcnyTestB.Step = 1 AND
        SC_P4_Etiketovacka.Step = 1 THEN
        P4_Pracovisko.STAV.READY:= TRUE;
    ELSE
        P4_Pracovisko.STAV.READY:= FALSE;
    END_IF

    //Zapnutie aspoň jedného Funkčného Testera//
    IF NOT P4_FunkcnyTestA.STAV.Tester_ON AND NOT P4_FunkcnyTestB.STAV.Tester_ON THEN
        P4_FunkcnyTestA.STAV.Tester_ON:= TRUE;
    END_IF

    //*******************************************Zapnutie osvetlenia pracoviska********************************//
    IF NOT Safety.IN.P4_PredneDvere_PritomPetlice THEN
        P4_Pracovisko.OUT.OsvetlenieBunky:= TRUE;
    ELSE
        P4_Pracovisko.OUT.OsvetlenieBunky:= FALSE;
    END_IF

    P4_Pracovisko.OUT.Osvetlenie_CAM15:= TRUE;
    P4_Pracovisko.OUT.Osvetlenie_CAM16:= TRUE;

    //****************************************Ovládanie majáka***********************************************//
    //Zelené svetlo//
    IF P4_Pracovisko.STAV.Automat THEN
        P4_Pracovisko.OUT.Majak_ZeleneSvetlo:= TRUE;
    ELSIF P4_Pracovisko.STAV.Manual THEN
        P4_Pracovisko.OUT.Majak_ZeleneSvetlo:= Blikac500ms;
    ELSE
        P4_Pracovisko.OUT.Majak_ZeleneSvetlo:= FALSE;
    END_IF

    //Žlté svetlo//
    IF P4_Pracovisko.STAV.Automat AND NOT P4_Pracovisko.STAV.PoINIT THEN
        P4_Pracovisko.OUT.Majak_ZlteSvetlo:= TRUE;
    ELSIF Linka.PAR.ZvolenyModel = '4F' AND NOT P4_FunkcnyTestA.IN.TypSpodnychKontaktov_4F THEN
        P4_Pracovisko.OUT.Majak_ZlteSvetlo:= Blikac500ms;
    ELSIF Linka.PAR.ZvolenyModel = '5F' AND NOT P4_FunkcnyTestA.IN.TypSpodnychKontaktov_5F_5H THEN
        P4_Pracovisko.OUT.Majak_ZlteSvetlo:= Blikac500ms;
    ELSIF Linka.PAR.ZvolenyModel = '5H' AND NOT P4_FunkcnyTestA.IN.TypSpodnychKontaktov_5F_5H THEN
        P4_Pracovisko.OUT.Majak_ZlteSvetlo:= Blikac500ms;
    ELSIF Linka.PAR.ZvolenyModel = '4F' AND NOT P4_FunkcnyTestB.IN.TypSpodnychKontaktov_4F THEN
        P4_Pracovisko.OUT.Majak_ZlteSvetlo:= Blikac500ms;
    ELSIF Linka.PAR.ZvolenyModel = '5F' AND NOT P4_FunkcnyTestB.IN.TypSpodnychKontaktov_5F_5H THEN
        P4_Pracovisko.OUT.Majak_ZlteSvetlo:= Blikac500ms;
    ELSIF Linka.PAR.ZvolenyModel = '5H' AND NOT P4_FunkcnyTestB.IN.TypSpodnychKontaktov_5F_5H THEN
        P4_Pracovisko.OUT.Majak_ZlteSvetlo:= Blikac500ms;
    ELSE
        P4_Pracovisko.OUT.Majak_ZlteSvetlo:= FALSE;
    END_IF

    //Červené svetlo//
    IF P4_Pracovisko.STAV.PORUCHA THEN
        P4_Pracovisko.OUT.Majak_CerveneSvetlo:= TRUE;
    ELSE
        P4_Pracovisko.OUT.Majak_CerveneSvetlo:= FALSE;
    END_IF

    //Zvuková signalizácia//
    //    IF EDGEPOS(P4_Pracovisko.STAV.PORUCHA) THEN
    //        P4_Pracovisko.OUT.Majak_Hukacka:= Blikac500ms;
    //    END_IF

    IF P34_AlarmyVizu.PotvrdAlarmy THEN
        P4_Pracovisko.OUT.Majak_Hukacka:= FALSE;
    END_IF

END_PROGRAM

PROGRAM _EXIT
	(* Insert code here *)

END_PROGRAM
```

#### OvlVentilovychTerminalov.st
```iecst
ACTION OvlVentilovychTerminalov:

		//Mapovanie ventilového terminálu - VT8//
	P4_Pracovisko.OUT.VT8_OUT1.0:= P4_FunkcnyTestA.OUT.ZasunStoper_YV163;
	P4_Pracovisko.OUT.VT8_OUT1.1:= P4_FunkcnyTestB.OUT.ZasunStoper_YV164;
	P4_Pracovisko.OUT.VT8_OUT1.2:= P4_Etiketovacka.OUT.ZasunStoper_YV165;
	P4_Pracovisko.OUT.VT8_OUT1.3:= P4_FunkcnyTestA.OUT.KontaktyTestera_VYSUN_YV171;
	P4_Pracovisko.OUT.VT8_OUT1.4:= P4_FunkcnyTestB.OUT.KontaktyTestera_VYSUN_YV172;
	P4_Pracovisko.OUT.VT8_OUT1.5:= P4_Etiketovacka.OUT.OfukEtikety_ZAPNI_YV174;
	P4_Pracovisko.OUT.VT8_OUT1.6:= P4_Etiketovacka.OUT.Aplikator_VYSUN_YV173;
	P4_Pracovisko.OUT.VT8_OUT1.7;

	P4_Pracovisko.OUT.VT8_OUT2.0:= P4_Etiketovacka.OUT.Prisavanie_ZAPNI_YV175;
	P4_Pracovisko.OUT.VT8_OUT2.1:= P4_Etiketovacka.OUT.Prisavanie_VYPNI_YV176;
	P4_Pracovisko.OUT.VT8_OUT2.2;
	P4_Pracovisko.OUT.VT8_OUT2.3;
	P4_Pracovisko.OUT.VT8_OUT2.4:= P4_Etiketovacka.OUT.VysunCentrovanie_YV166;
	P4_Pracovisko.OUT.VT8_OUT2.5:= P4_Etiketovacka.OUT.ZasunCentrovanie_YV167;
	P4_Pracovisko.OUT.VT8_OUT2.6;
	P4_Pracovisko.OUT.VT8_OUT2.7;

	P4_Pracovisko.OUT.VT8_OUT3.0:= P4_FunkcnyTestA.OUT.HorneKontakty_ZASUN_YV177;
	P4_Pracovisko.OUT.VT8_OUT3.1:= P4_FunkcnyTestA.OUT.HorneKontakty_VYSUN_YV178;
	P4_Pracovisko.OUT.VT8_OUT3.2:= P4_FunkcnyTestA.OUT.OdpruzenieKontaktov_ZAPNI_YV179;
	P4_Pracovisko.OUT.VT8_OUT3.3:= P4_FunkcnyTestA.OUT.OdpruzenieKontaktov_VYPNI_YV180;
	P4_Pracovisko.OUT.VT8_OUT3.4:= P4_FunkcnyTestA.OUT.VysunCentrovanie_YV183;
	P4_Pracovisko.OUT.VT8_OUT3.5:= P4_FunkcnyTestA.OUT.ZasunCentrovanie_YV184;
	P4_Pracovisko.OUT.VT8_OUT3.6:= P4_FunkcnyTestA.OUT.SpodneKontakty_ZASUN_YV181;
	P4_Pracovisko.OUT.VT8_OUT3.7:= P4_FunkcnyTestA.OUT.SpodneKontakty_VYSUN_YV182;

	P4_Pracovisko.OUT.VT8_OUT4.0:= P4_FunkcnyTestB.OUT.HorneKontakty_ZASUN_YV185;
	P4_Pracovisko.OUT.VT8_OUT4.1:= P4_FunkcnyTestB.OUT.HorneKontakty_VYSUN_YV186;
	P4_Pracovisko.OUT.VT8_OUT4.2:= P4_FunkcnyTestB.OUT.OdpruzenieKontaktov_ZAPNI_YV187;
	P4_Pracovisko.OUT.VT8_OUT4.3:= P4_FunkcnyTestB.OUT.OdpruzenieKontaktov_VYPNI_YV188;
	P4_Pracovisko.OUT.VT8_OUT4.4:= P4_FunkcnyTestB.OUT.VysunCentrovanie_YV191;
	P4_Pracovisko.OUT.VT8_OUT4.5:= P4_FunkcnyTestB.OUT.ZasunCentrovanie_YV192;
	P4_Pracovisko.OUT.VT8_OUT4.6:= P4_FunkcnyTestB.OUT.SpodneKontakty_ZASUN_YV189;
	P4_Pracovisko.OUT.VT8_OUT4.7:= P4_FunkcnyTestB.OUT.SpodneKontakty_VYSUN_YV190;

END_ACTION
```

#### ProfinetKomunikaciaKAM14.st
```iecst
ACTION ProfinetKomunikaciaKAM14:

	CAM14.STAV.READY;

	//Vstupy pre kameru//
	CAM14.Profinet_PLC_OUTPUTS[0].0:= CAM14.CMD.Triger;

	//Výstupy z kamery//
	CAM14.STAV.SWITCH:= CAM14.Profinet_PLC_INPUTS[10].0;

	//Výsledky kamery//
	CAM14.RESULT.PowerCP.CitanieQRkodu_PowerCP_OK:= CAM14.Profinet_PLC_INPUTS[4].0;

	//Prečítaný QR kód DPS//
	IF EDGE(CAM14.STAV.SWITCH) THEN
		brsstrcpy(ADR(CAM14.RESULT.PowerCP.PrecitanyQRkod_PowerCP),ADR(CAM14.Profinet_QRkod_Znaky));
	END_IF

	//Stav výsledky READY//
	IF EDGE(CAM14.STAV.SWITCH)THEN
		CAM14.STAV.Results_READY:= TRUE;
	END_IF

END_ACTION
```

#### ProfinetKomunikaciaKAM15.st
```iecst
ACTION ProfinetKomunikaciaKAM15:

	//Vstupy pre kameru//
	CAM15.Profinet_PLC_OUTPUTS[0].3:= CAM15.CMD.Triger;

	//Výstupy z kamery//
	CAM15.STAV.READY:= CAM15.Profinet_PLC_INPUTS[0].0;
	CAM15.STAV.SWITCH:= CAM15.Profinet_PLC_INPUTS[0].1;
    CAM15.STAV.BUSY:= CAM15.Profinet_PLC_INPUTS[0].2;
    CAM15.STAV.Command_AKCEPTOVANY:= CAM15.Profinet_PLC_INPUTS[0].3;
    CAM15.STAV.Command_READY:= CAM15.Profinet_PLC_INPUTS[0].4;
    CAM15.STAV.Command_ERROR:= CAM15.Profinet_PLC_INPUTS[0].5;

	//Výsledky kamery//

	//Výsledky kamery//
	CAM15.RESULT.CitanieQRkodu_Etikety_OK:= CAM15.Profinet_PLC_INPUTS[2].0;
	CAM15.RESULT.Pritomn_Etikety:= CAM15.Profinet_PLC_INPUTS[2].1;
	CAM15.RESULT.Pritomn_LogoBMV:= CAM15.Profinet_PLC_INPUTS[2].2;
	CAM15.RESULT.Pritomn_Textu_PowerCP:= CAM15.Profinet_PLC_INPUTS[2].3;
	CAM15.RESULT.Pritomn_Textu_Panasonic:= CAM15.Profinet_PLC_INPUTS[2].4;
	CAM15.RESULT.Pritomn_Textu_SK:= CAM15.Profinet_PLC_INPUTS[2].5;

	//Prečítaný QR kód etikety a OCR etikety//
	IF EDGE(CAM15.STAV.SWITCH) THEN
		brsstrcpy(ADR(CAM15.RESULT.PrecitanyQRkod_Etikety),ADR(CAM15.Profinet_QRkod_Znaky));
		brsstrcpy(ADR(CAM15.RESULT.PrecitaneOCR_Etikety),ADR(CAM15.Profinet_OCR_Znaky));
	END_IF

	//Stav výsledky READY//
	IF EDGE(CAM15.STAV.SWITCH)THEN
		CAM15.STAV.Results_READY:= TRUE;
	END_IF

END_ACTION
```

#### ProfinetKomunikaciaKAM16.st
```iecst
ACTION ProfinetKomunikaciaKAM16:

	//Vstupy pre kameru//
	CAM16.Profinet_PLC_OUTPUTS[0].3:= CAM16.CMD.Triger;

	//Výstupy z kamery//
	CAM16.STAV.READY:= CAM16.Profinet_PLC_INPUTS[0].0;
	CAM16.STAV.SWITCH:= CAM16.Profinet_PLC_INPUTS[0].1;
    CAM16.STAV.BUSY:= CAM16.Profinet_PLC_INPUTS[0].2;
    CAM16.STAV.Command_AKCEPTOVANY:= CAM16.Profinet_PLC_INPUTS[0].3;
    CAM16.STAV.Command_READY:= CAM16.Profinet_PLC_INPUTS[0].4;
    CAM16.STAV.Command_ERROR:= CAM16.Profinet_PLC_INPUTS[0].5;

	//Výsledky kamery//
	CAM16.RESULT.Paletka.Pritomn_Busbarov_4F:= CAM16.Profinet_PLC_INPUTS[2].0;
	CAM16.RESULT.Paletka.Pritomn_Busbarov_5F:= CAM16.Profinet_PLC_INPUTS[2].1;
	CAM16.RESULT.Paletka.Pritomn_Busbarov_5H:= CAM16.Profinet_PLC_INPUTS[2].2;
	CAM16.RESULT.Paletka.Pritomn_LavyMVcase:= CAM16.Profinet_PLC_INPUTS[2].3;
	CAM16.RESULT.Paletka.Pritomn_PravyMVcase:= CAM16.Profinet_PLC_INPUTS[2].4;
    CAM16.RESULT.Paletka.Pritomn_PowerCP:= CAM16.Profinet_PLC_INPUTS[2].5;
    CAM16.RESULT.PowerCP.PritomnostSkrutky_K40:= CAM16.Profinet_PLC_INPUTS[2].7;

    CAM16.RESULT.PowerCP.PritomnostSkrutky_M5:= CAM16.Profinet_PLC_INPUTS[3].0;

	//Stav výsledky READY//
	IF EDGE(CAM16.STAV.SWITCH)THEN
		CAM16.STAV.Results_READY:= TRUE;
	END_IF

END_ACTION
```

### Program Logical/Program/Pracovisko_4/P4_Dopravniky (IEC)

#### Main.st - Init, cyclic, exit code
```iecst
PROGRAM _INIT
	(* Insert code here *)

END_PROGRAM

PROGRAM _CYCLIC

	//Volanie funkcie SequenceControl//
	SequenceControl(SC:= SC_P4_Dopravniky);

	//Reset sekcie //
    IF NOT Safety.STAV.P4_ZonaBunky_AKTIVNA THEN
        SC_P4_Dopravniky.Step:= 0;
    ELSIF P4_Dopravniky.Reset THEN
		SC_P4_Dopravniky.Step:= 0;
		P4_Dopravniky.Reset:= FALSE;
	END_IF

	CASE SC_P4_Dopravniky.Step OF

		0:
			SC_P4_Dopravniky.StepName:='0 - Nulovanie';
			P4_Dopravniky.Automat:= FALSE;
			P4_Dopravniky.KoniecCyklu:= FALSE;
			P4_Dopravniky.Manual:= FALSE;
			P4_Dopravniky.STAV.PoINIT:= FALSE;
			P4_Dopravniky.OUT.HornyDoprav_ChodVPRED_M24:= FALSE;
			P4_Dopravniky.OUT.SpodnyDoprav_ChodVPRED_M27:= FALSE;

			IF Safety.STAV.P4_ZonaBunky_AKTIVNA AND NOT P4_Pracovisko.STAV.PORUCHA AND P4_Pracovisko.IN.PrivodVzduchu_SnimacTlaku_S15 THEN
				SC_P4_Dopravniky.ResetStep:= TRUE;
				SC_P4_Dopravniky.Step:= 1;
			END_IF

		1:
			SC_P4_Dopravniky.StepName:='1 - Cakam na spustenie vyroby';
			P4_Dopravniky.KoniecCyklu:= FALSE;
            IF P4_Dopravniky.Automat THEN
				SC_P4_Dopravniky.Step:= 2;
			ELSIF P4_Dopravniky.Manual THEN
				SC_P4_Dopravniky.Step:= 700;
			END_IF

			//********************************************************Inicializácia****************************************************************************//

		2:
			SC_P4_Dopravniky.StepName:='2 - Inicializacia - cakam na spustenie inicializacie';
			SC_P4_Dopravniky.IdleTime.PT:= T#2s;
			SC_P4_Dopravniky.AlarmTime.PT:= T#5s;

			IF P4_FunkcnyTestA_VychodziaPozicia AND P4_FunkcnyTestB_VychodziaPozicia (*AND P4_Etiketovacka_VychodziaPozicia*) THEN
				SC_P4_Dopravniky.IdleTime.IN:= TRUE;
			ELSE
				SC_P4_Dopravniky.IdleTime.IN:= FALSE;
			END_IF

			IF SC_P4_Dopravniky.IdleTime.Q THEN
				SC_P4_Dopravniky.ResetStep:= TRUE;
				SC_P4_Dopravniky.Step:= 3;
			END_IF

		3:
			SC_P4_Dopravniky.StepName:='2 - Inicializacia - ukoncenie inicializacie';
			SC_P4_Dopravniky.IdleTime.PT:= T#4s;
			SC_P4_Dopravniky.AlarmTime.PT:= T#5s;

			P4_Dopravniky.OUT.HornyDoprav_ChodVPRED_M24:= TRUE;
			P4_Dopravniky.OUT.SpodnyDoprav_ChodVPRED_M27:= TRUE;
			SC_P4_Dopravniky.IdleTime.IN:= TRUE;

			IF SC_P4_Dopravniky.IdleTime.Q THEN
				P4_Dopravniky.STAV.PoINIT:= TRUE;
				SC_P4_Dopravniky.ResetStep:= TRUE;
				SC_P4_Dopravniky.Step:= 100;
			END_IF

			//********************************************************Automatický režim****************************************************************************//
		100:
			SC_P4_Dopravniky.StepName:='100 - Automaticky Rezim - cakam na vypnutie dopravnikou';
			SC_P4_Dopravniky.IdleTime.PT:= T#200ms;
			SC_P4_Dopravniky.AlarmTime.PT:= T#5s;

			IF P4_Dopravniky.KoniecCyklu AND NOT P4_FunkcnyTestA.Automat AND NOT P4_FunkcnyTestB.Automat AND NOT P4_Etiketovacka.Automat AND Safety.STAV.P3_VystupBunky_Bariera_AKTIVNA AND Safety.STAV.P4_VystupBunky_Bariera_AKTIVNA THEN
				SC_P4_Dopravniky.ResetStep:= TRUE;
				SC_P4_Dopravniky.Step:= 0;
			END_IF

			//*******************************************************Manuálny režim*******************************************************************************//
		700:
			SC_P4_Dopravniky.StepName:='700 - Manualny Rezim';
			SC_P4_Dopravniky.IdleTime.PT:= T#8s;
			SC_P4_Dopravniky.AlarmTime.PT:= T#5s;

	END_CASE

END_PROGRAM

PROGRAM _EXIT
	(* Insert code here *)

END_PROGRAM
```

### Program Logical/Program/Pracovisko_4/P4_Vytah (IEC)
